# EPICS substitutions: bsaDriverApp/Db/bsssCtrl_localTest.substitutions
file serviceControl.db {
    pattern {   DEVICE,   SERVICE }
            { "$(DEV)" ,  "BSSS"}
}

file bsssRateLimit_localTest.db {
    pattern {   DEVICE,   SERVICE }
            { "$(DEV)" ,  "BSSS"}
}

file serviceStatus.db {
    pattern {   DEVICE,    SERVICE }
            { "$(DEV)" ,  "BSSS0"}
            { "$(DEV)" ,  "BSSS1"}

}
